PROGRAM prgAddedProperties
VAR
	{attribute addProperty Name "X"}
	fbDriveX : fbDrive;
	
	{attribute addProperty Name "Y"}
	fbDriveY : fbDrive;
	
	{attribute addProperty Name "Z"}
	fbDriveZ : fbDrive;
END_VAR

fbDriveX();
fbDriveY();
fbDriveZ();

END_PROGRAM

(* stored: Version 1.1.0.1, ProductVersion 3.1.4024.2
   POU prgAddedProperties: Id {c9b6b6b5-de79-4a8c-ae2c-3902dd66ffac}, SpecialFunc None *)
